FUNCTION_BLOCK FB_FindTextIndexNum
VAR_INPUT
	iText:T_MaxString;
	
END_VAR
VAR_OUTPUT
	
	qIndexNum: INT;
	qLineIsValid: BOOL;


END_VAR
VAR
		textidNameLocation: INT;
		textIDlocname: STRING(255);
		isTextIDLinee: BOOL;
		textidline: INT;
isTextIDLine: BOOL;
textIDnameLefted: STRING(255);
textidline2: INT;
	textlen: INT;
	
	textidline3: STRING(255);

END_VAR
VAR // added by the converter: edge detectors and wires of the graphical bodies
    _w1, _w2 : BOOL;
END_VAR

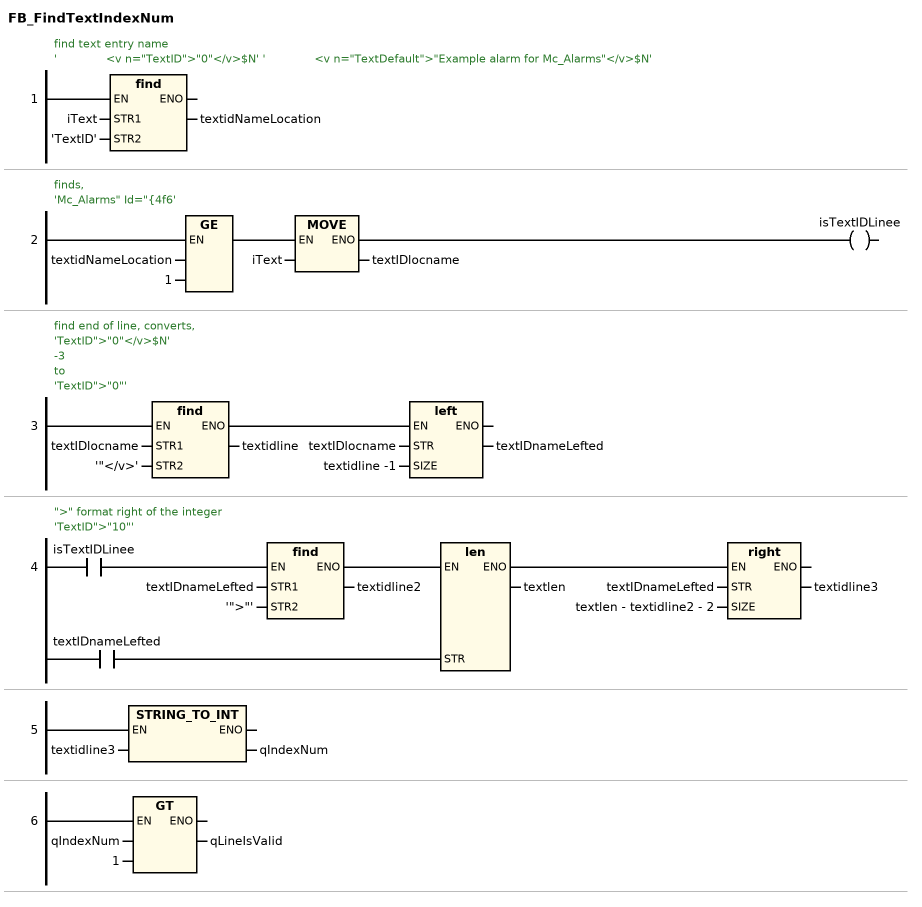
// NETWORK 1
// find text entry name
// '              <v n="TextID">"0"</v>$N' '              <v n="TextDefault">"Example alarm for Mc_Alarms"</v>$N'
textidNameLocation := find(STR1 := iText, STR2 := 'TextID');

// NETWORK 2
// finds,
// 'Mc_Alarms" Id="{4f6'
_w1 := textidNameLocation >= 1;
IF _w1 THEN textIDlocname := iText; END_IF
isTextIDLinee := _w1;

// NETWORK 3
// find end of line, converts,
// 'TextID">"0"</v>$N'
// -3
// to
// 'TextID">"0"'
textidline := find(STR1 := textIDlocname, STR2 := '"</v>');
textIDnameLefted := left(STR := textIDlocname, SIZE := textidline -1);

// NETWORK 4
// ">" format right of the integer
//
// 'TextID">"10"'
_w2 := isTextIDLinee;
IF _w2 THEN textidline2 := find(STR1 := textIDnameLefted, STR2 := '">"'); END_IF
IF _w2 THEN textlen := len(STR := textIDnameLefted); END_IF
IF _w2 THEN textidline3 := right(STR := textIDnameLefted, SIZE := textlen - textidline2 - 2); END_IF

// NETWORK 5
qIndexNum := STRING_TO_INT(textidline3);

// NETWORK 6
qLineIsValid := qIndexNum > 1;

END_FUNCTION_BLOCK

(* stored: Version 1.1.0.1, ProductVersion 3.1.4024.12
   POU FB_FindTextIndexNum: Id {d63743f3-2eb0-408c-a75d-1e453a846348}, SpecialFunc None *)
